PROGRAM MAIN
VAR
END_VAR

END_PROGRAM

(* stored: Version 1.1.0.1, ProductVersion 3.1.0.36
   POU MAIN: Id {3384ea04-753c-49b9-9a80-72d1c4f3cd9d} *)
